// Mitsubishi GX Works2 project: GX W2 L2 Ex 4 DK c   PLC: FX3G

// global labels: Global1
VAR_GLOBAL
  iStartSyst_PB AT X001 : BOOL;
  iStop_PB AT Y001 : BOOL;
  oFillValve AT Y001 : BOOL;
END_VAR

// task Task_01 (event TRUE, interval 0, priority 31): POU_01

PROGRAM POU_01
VAR
  iSystem_Started : BOOL;
  RetentiveTimer_1 : TIMER_CONT_FB_M;
  RetentiveTimer_1_ElapsedTime : INT;
  RetentiveTimer_1_Done : BOOL;
END_VAR
(* structured ladder/FBD written out as ST: instructions are called as NAME(EN, inputs, outputs); _pN, _eN, _tN stand for wires *)
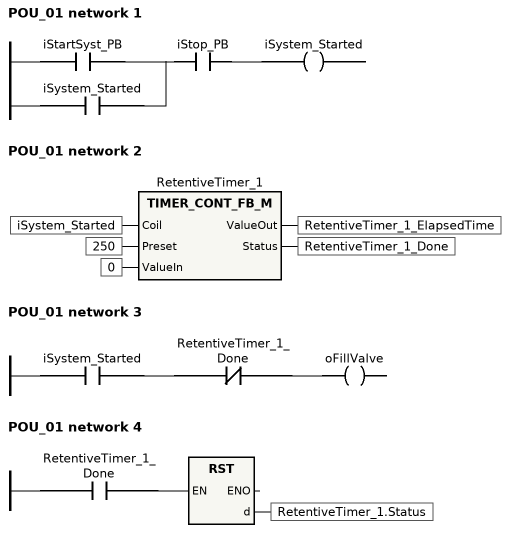
(* network 1 *)
iSystem_Started := (iStartSyst_PB OR iSystem_Started) AND iStop_PB;
(* network 2 *)
RetentiveTimer_1(Coil := iSystem_Started, Preset := 250, ValueIn := 0, ValueOut => RetentiveTimer_1_ElapsedTime, Status => RetentiveTimer_1_Done);
(* network 3 *)
oFillValve := iSystem_Started AND NOT RetentiveTimer_1_Done;
(* network 4 *)
RST(RetentiveTimer_1_Done, RetentiveTimer_1.Status);
END_PROGRAM
